FUNCTION F_GetTU_PresentStateEmulation : BOOL
(**************************************************************************************
 * 	Application		:	BoxControl Framework
 *	Revision		:	$Revision: 404529 $
 *	Revision date	:	$Date: 2018-04-23 08:21:38 +0200 (Mo., 23 Apr 2018) $
 *	Last changed by	:	$Author: b7bolm $
 *	URL				:	$URL: http://almscdc.swisslog.com/repo/SWPD/Development/BoxControlFramework/20_Release/trunk/01_Software/BCF/BCF/JumpStart/20_Product/11_Emu/12_E_Functions/10_Lib/10_Conv/10_Functions/F_GetTU_PresentStateEmulation.TcPOU $
 *
 *	Purpose			:	Returns TU present state
 *
 * ------------------------------------------------------------------------------------
 *	Copyright Swisslog [IP AG], Switzerland. All rights reserved.
 * 
 * ------------------------------------------------------------------------------------
 *	
 * 	Revision History: 
 *
 * 	VERSION			DATE			INITIALS			DESCRIPTION
 *	0.1				01.01.2001		swl					Example
 *
 **************************************************************************************)
VAR_INPUT
	eFunctionNumber	: E_FunctionNumber; // Function number of corresponding function
	ZoneNumber 		: INT; // Zone number
	Position        : UINT;
END_VAR


VAR_OUTPUT
	TU_DataIndex 	: DINT;	
END_VAR

// Check if function number is valid
IF eFunctionNumber > E_FunctionNumber.F_BEGIN_FUNCTION AND
   eFunctionNumber < E_FunctionNumber.F_END_FUNCTION THEN

	// Check reference is valid
	IF __ISVALIDREF(FunctionRegistryEmulation[eFunctionNumber].rFunction) THEN
   		// Return TU present state
   		F_GetTU_PresentStateEmulation := FunctionRegistryEmulation[eFunctionNumber].rFunction.M_GetTU_PresentState(
																	mZone := ZoneNumber,
																	mPosition := Position,
																	mTU_DataIndex => TU_DataIndex);
	END_IF
END_IF

END_FUNCTION

(* stored: Version 1.1.0.1, ProductVersion 3.1.4022.12
   POU F_GetTU_PresentStateEmulation: Id {acf5c546-3f28-4066-99d4-73c4dfd46bea}, SpecialFunc None *)
